DATA_BLOCK "开关门控制_DB"
{ S7_Optimized_Access := 'TRUE' }
VERSION : 0.1
NON_RETAIN
"开关门控制"

BEGIN

END_DATA_BLOCK

